TYPE ST_AxisControlManualHMI :
STRUCT
	bEnableManualMode							: BOOL;
	bConsequentialError							: BOOL;
	bError										: BOOL;
	nErrorID									: UDINT;
	fSetPos										: LREAL;					// Set position (absolut value from NC)
	fModuloSetPos								: LREAL;					// Actual modulo position (absolut value from NC)
	fSetVelo									: LREAL;					// Set velocity
	fSetTorque									: LREAL;
	fActPos										: LREAL;					// Actual position (absolut value from NC)
	fModuloActPos								: LREAL;					// Actual modulo position (absolut value from NC)
	fActVelo									: LREAL;					// Actual velocity
	fActTorque									: LREAL;
	fPosDiff									: LREAL;					// Position difference (lag distance)
	stCommands									: ST_AxisControlManual;
	stStatus									: REFERENCE TO Tc2_MC2.ST_AxisStatus;
	stParameters								: REFERENCE TO Tc2_MC2.ST_AxisParameterSet;
END_STRUCT
END_TYPE

(* stored: Version 1.2.0.0, ProductVersion 3.1.4026.13, FileIdentifier c4226aa18327e21b5e94803ce79eac1d9fcf64c4, FileSignature 799a33f412f5bae2ab33fbd60435bf0eb5c4d6c62819c0bd9cd3373b3413b3f0e58069834c950359ceac13cd8d365fbbf5ed8075b29e6a4a8e8871b149595befd37f44dba51c9ce86428cf48e6d4d67ace79d9eaec7bc45cb853380d0ab47cd81519becef393c08a56eb058880e03ecc03e0da69f4561b4f8e4e7e8866486c89d763119bf7505c15c680e04d39ccbecf0da78570ed73112bc2e02a7b6eea8cbfc826ecc4aab4d970ba111476f1ddca50e8c4e7581d3cdfb663265dab82a034a0c0943dad3687da3bbc8bf51d84761b5fd15d87291369f7e6c323605bdf89b3c1c8d8e4379ee9e8f2b336f14b0869c0b80f2e38c7a53bd98edfcf9aa4035e5444
   DUT ST_AxisControlManualHMI: Id {17433bbb-ba3a-4950-94b2-37b635d90cd5} *)
